PROGRAM MAIN
VAR
	fbRpc		: tchaxx.FB_RPC(sAmsNetId:= tchaxx.GCL.cLocalAmsNetId, nAmsPort:= 852, sInstancePath:= 'MAIN.fbRpcServer', sSymbol:= 'Greet');
	
	// Arguments and RetVal
	sArg  : T_MaxString := _AppInfo.AppName;
	nLen  : INT;
	stLibVersion : ST_LibVersion := Tc3_Module.Global_Version.stLibVersion_Tc3_Module;
	sRetVal : T_MaxString;
	stRetVal : ST_AdsStatus;
END_VAR


stRetVal := fbRpc.VarInput(sArg)
                 .VarOutput(nLen)
                 .VarInOut(stLibVersion)
                 .ReturnValue(sRetVal)
                 .Invoke();

END_PROGRAM

(* stored: Version 1.1.0.1, ProductVersion 3.1.4024.12
   POU MAIN: Id {b3812910-b416-492a-aa5d-1cfbbaf30e41}, SpecialFunc None *)
